// TwinCAT 3 PLC project Pinana
// Title: Pinanas
// Company: ekvip automation GmbH
// Author: Ajnin and Yeknom
// Description: short summary ============= This project was created for the YouTube channel https://www.youtube.com/@ninjamonkeystutorials created. It is intended to show why references as return values for functions are dangerous. legal notes ======== SPDX-FileCopyrightText: © 2024 ekvip automation GmbH <info@ekvip.de> SPDX-License-Identifier: Apache-2.0 For details check: Apache-2.0_
// ProgramVersion: 3.1.4024.0
// libraries:
//   Tc2_Standard, * (Beckhoff Automation GmbH)
//   Tc2_System, * (Beckhoff Automation GmbH)
//   Tc3_Module, * (Beckhoff Automation GmbH)
// project tree:
//   Pinana/Banana/Types/Enums/ BananaType.TcDUT
//   Pinana/Functions/ CalculatePinanaCurvature.TcPOU, GetANewPinana.TcPOU, GetAPinana.TcPOU, GetAPinanaFromGlobal.TcPOU, GetAPinanaFromStack.TcPOU, IsSetPinanaCallByRef.TcPOU
//   Pinana/GVLs/ PinanaPrototypes.TcGVL
//   Pinana/Pineapple/Types/Enums/ PineappleType.TcDUT
//   Pinana/Types/Enums/ PinanaType.TcDUT
//   Pinana/Types/Structures/ Pinana.TcDUT
//   Tasks/main/ MAIN.TcPOU, PlcTask.TcTTO
// real-time tasks:
//   TASK PlcTask: cycle T#10ms, priority 20, ADS port 350

CONFIGURATION Pinana
    RESOURCE PLC ON TwinCAT3
        TASK PlcTask(INTERVAL := T#10ms, PRIORITY := 20);
        PROGRAM MAIN WITH PlcTask : MAIN;
    END_RESOURCE
END_CONFIGURATION

// ---- Pinana/Banana/Types/Enums/BananaType.TcDUT
(*

short summary
=============
This enumeration represents the banana varieties from which π-nana are to be produced.
If the type is extended, make sure that only the least significant nibble is used.
Only 15 banana types can be mapped, namely from 16#01 to 16#0F.
The software generates the π-nana type by adding the pineapple type and the banana type.
So that everything remains unique, the pineapple variety is given the second nibble from 16#10 to 16#F0.

legal notes
===========
SPDX-FileCopyrightText: © 2024 ekvip automation GmbH <info@ekvip.de>
SPDX-License-Identifier: Apache-2.0
For details check: Apache-2.0_

.. _Apache-2.0: https://www.apache.org/licenses/LICENSE-2.0

*)
{attribute 'qualified_only'}
{attribute 'strict'}
{attribute 'to_string'}
TYPE BananaType :(
	(* it's not a banana *)
	NONE		:= 16#00,
	(* it's a cavendish banana *)
	CAVENDISH	:= 16#01,
	(* it's a plaintain banana *)
	PLANTAIN	:= 16#02,
	(* it's a red banana *)
	RED_BANANA	:= 16#03,
	(* it's a lady finger banana and not an okra *)
	LADY_FINGER	:= 16#04
)UDINT := NONE;
END_TYPE

// ---- Pinana/Pineapple/Types/Enums/PineappleType.TcDUT
(*

short summary
=============
This enumeration represents the pineapple varieties from which π-nana are to be produced.
If the type is extended, make sure that only the second nibble is used.
Only 15 pineapple types can be mapped, namely from 16#10 to 16#F0.
The software generates the π-nana type by adding the pineapple type and the banana type.
So that everything remains unique, the banana variety is given the least significant nibble from 16#01 to 16#0F.


legal notes
===========
SPDX-FileCopyrightText: © 2024 ekvip automation GmbH <info@ekvip.de>
SPDX-License-Identifier: Apache-2.0
For details check: Apache-2.0_

.. _Apache-2.0: https://www.apache.org/licenses/LICENSE-2.0

*)
{attribute 'qualified_only'}
{attribute 'strict'}
{attribute 'to_string'}
TYPE PineappleType :(
	(* it's not a pineapple *)
	NONE		:= 16#00,
	(* it's an abacaxi pineapple *)
	ABACAXI		:= 16#10,
	(* it's a queen pineapple *)
	QUEEN		:= 16#20,
	(* it's a mordilona pineapple *)
	MORDILONA	:= 16#30,
	(* it's a panare pineapple *)
	PANARE		:= 16#40
)UDINT := NONE;
END_TYPE

// ---- Pinana/Types/Enums/PinanaType.TcDUT
(*

short summary
=============
This enumeration represents the π-nana types.
The type of π-nana is determined by the simple formula
π-nana type := pineapple type + banana type 

legal notes
===========
SPDX-FileCopyrightText: © 2024 ekvip automation GmbH <info@ekvip.de>
SPDX-License-Identifier: Apache-2.0
For details check: Apache-2.0_

.. _Apache-2.0: https://www.apache.org/licenses/LICENSE-2.0

*)
{attribute 'qualified_only'}
{attribute 'to_string'}
TYPE PinanaType :
(
	(* it's not a pinana *)
	NONE		:= 16#00,
	(* PineappleType.ABACAXI + BananaType.CAVENDISH *)
	ABADISH 	:= 16#11,
	(* PineappleType.ABACAXI + BananaType.PLANTAIN *)
	PLANABA		:= 16#12,
	(* PineappleType.ABACAXI + BananaType.RED_BANANA *)
	ABANANA		:= 16#13,
	(* PineappleType.ABACAXI + BananaType.LADY_FINGER *)
	ABA_LADY	:= 16#14,
	(* PineappleType.QUEEN + BananaType.CAVENDISH *)
	CAVEEN	 	:= 16#21,
	(* PineappleType.QUEEN + BananaType.PLANTAIN *)
	PLEEN		:= 16#22,
	(* PineappleType.QUEEN + BananaType.RED_BANANA *)
	RED_QUEEN	:= 16#23,
	(* PineappleType.QUEEN + BananaType.LADY_FINGER *)
	LADY_QUEEN	:= 16#24,
	(* PineappleType.MORDILONA + BananaType.CAVENDISH *)
	ILONACAVE 	:= 16#31,
	(* PineappleType.MORDILONA + BananaType.PLANTAIN *)
	PLAONA		:= 16#32,
	(* PineappleType.MORDILONA + BananaType.RED_BANANA *)
	RED_LONA	:= 16#33,
	(* PineappleType.MORDILONA + BananaType.LADY_FINGER *)
	LADY_LONA	:= 16#34,
	(* PineappleType.PANARE + BananaType.CAVENDISH *)
	PANDISH 	:= 16#41,
	(* PineappleType.PANARE + BananaType.PLANTAIN *)
	PLANPAN		:= 16#42,
	(* PineappleType.PANARE + BananaType.RED_BANANA *)
	PANANA		:= 16#43,
	(* PineappleType.PANARE + BananaType.LADY_FINGER *)
	PAN_FINGER	:= 16#44	
)UDINT := NONE;
END_TYPE

// ---- Pinana/Types/Structures/Pinana.TcDUT
(*

short summary
=============
This type struct contains the properties of a π-nana.

legal notes
===========
SPDX-FileCopyrightText: © 2024 ekvip automation GmbH <info@ekvip.de>
SPDX-License-Identifier: Apache-2.0
For details check: Apache-2.0_

.. _Apache-2.0: https://www.apache.org/licenses/LICENSE-2.0

*)
TYPE Pinana :
STRUCT
	(* pointer to itself for destruction of dynamically created Pinanas *)
	me			:POINTER TO Pinana := 0;
	(* type of π-nana *)
	pinanaType	:PinanaType;
	(* name of the π-nana variety *)
	variety		:STRING;
	(* curvature of π-nana ofcourse in radians *)
	curve		:LREAL;
END_STRUCT
END_TYPE

// ---- Pinana/GVLs/PinanaPrototypes.TcGVL
(*

short summary
=============
This is a lookup table for π-nanas.
It's not a constant because the function GetAPinanaFromGlobal
has a reference to π-nana as return value. A reference requires write access.

The attribute hide is not used because we want show it online how to screw it. 

legal notes
===========
SPDX-FileCopyrightText: © 2024 ekvip automation GmbH <info@ekvip.de>
SPDX-License-Identifier: Apache-2.0
For details check: Apache-2.0_

.. _Apache-2.0: https://www.apache.org/licenses/LICENSE-2.0

*)
{attribute 'qualified_only'}
VAR_GLOBAL
	(* lookup table for π-nanas *)
	pinanas :ARRAY[
		SHR(PineappleType.ABACAXI,4)..SHR(PineappleType.PANARE,4)
	] OF ARRAY[
		BananaType.CAVENDISH..BananaType.LADY_FINGER
	] OF Pinana := [
		[
			(pinanaType := PinanaType.ABADISH,		variety := TO_STRING(PinanaType.ABADISH),	curve := CalculatePinanaCurvature(PinanaType.ABADISH),		me := ADR(pinanas[1][1])),
			(pinanaType := PinanaType.PLANABA,		variety := TO_STRING(PinanaType.PLANABA),	curve := CalculatePinanaCurvature(PinanaType.PLANABA),		me := ADR(pinanas[1][2])),
			(pinanaType := PinanaType.ABANANA,		variety := TO_STRING(PinanaType.ABANANA),	curve := CalculatePinanaCurvature(PinanaType.ABANANA),		me := ADR(pinanas[1][3])),
			(pinanaType := PinanaType.ABA_LADY,		variety := TO_STRING(PinanaType.ABA_LADY),	curve := CalculatePinanaCurvature(PinanaType.ABA_LADY),		me := ADR(pinanas[1][4]))
		],[
			(pinanaType := PinanaType.CAVEEN,		variety := TO_STRING(PinanaType.CAVEEN),	curve := CalculatePinanaCurvature(PinanaType.CAVEEN),		me := ADR(pinanas[2][1])),
			(pinanaType := PinanaType.PLEEN,		variety := TO_STRING(PinanaType.PLEEN),		curve := CalculatePinanaCurvature(PinanaType.PLEEN),		me := ADR(pinanas[2][2])),
			(pinanaType := PinanaType.RED_QUEEN,	variety := TO_STRING(PinanaType.RED_QUEEN),	curve := CalculatePinanaCurvature(PinanaType.RED_QUEEN),	me := ADR(pinanas[2][3])),
			(pinanaType := PinanaType.LADY_QUEEN,	variety := TO_STRING(PinanaType.LADY_QUEEN),curve := CalculatePinanaCurvature(PinanaType.LADY_QUEEN),	me := ADR(pinanas[2][4]))
		],[
			(pinanaType := PinanaType.ILONACAVE,	variety := TO_STRING(PinanaType.ILONACAVE),	curve := CalculatePinanaCurvature(PinanaType.ILONACAVE),	me := ADR(pinanas[3][1])),
			(pinanaType := PinanaType.PLAONA,		variety := TO_STRING(PinanaType.PLAONA),	curve := CalculatePinanaCurvature(PinanaType.PLAONA),		me := ADR(pinanas[3][2])),
			(pinanaType := PinanaType.RED_LONA,		variety := TO_STRING(PinanaType.RED_LONA),	curve := CalculatePinanaCurvature(PinanaType.RED_LONA),		me := ADR(pinanas[3][3])),
			(pinanaType := PinanaType.LADY_LONA,	variety := TO_STRING(PinanaType.LADY_LONA),	curve := CalculatePinanaCurvature(PinanaType.LADY_LONA),	me := ADR(pinanas[3][4]))
		],[
			(pinanaType := PinanaType.PANDISH,		variety := TO_STRING(PinanaType.PANDISH),	curve := CalculatePinanaCurvature(PinanaType.PANDISH),		me := ADR(pinanas[4][1])),
			(pinanaType := PinanaType.PLANPAN,		variety := TO_STRING(PinanaType.PLANPAN),	curve := CalculatePinanaCurvature(PinanaType.PLANPAN),		me := ADR(pinanas[4][2])),
			(pinanaType := PinanaType.PANANA,		variety := TO_STRING(PinanaType.PANANA),	curve := CalculatePinanaCurvature(PinanaType.PANANA),		me := ADR(pinanas[4][3])),
			(pinanaType := PinanaType.PAN_FINGER,	variety := TO_STRING(PinanaType.PAN_FINGER),curve := CalculatePinanaCurvature(PinanaType.PAN_FINGER),	me := ADR(pinanas[4][4]))
		]
	];
END_VAR

// ---- Tasks/main/MAIN.TcPOU
(*

short summary
=============
This program is attached to the main plc task.
This project was created for the YouTube channel https://www.youtube.com/@ninjamonkeystutorials
created. It is intended to show why references as return values for functions are dangerous.
You've a couple of flags to control the data flow... 
It can be a lot of fun to mess with TwinCAT, if it's not a real world plc. So have fun with it.

legal notes
===========
SPDX-FileCopyrightText: © 2024 ekvip automation GmbH <info@ekvip.de>
SPDX-License-Identifier: Apache-2.0
For details check: Apache-2.0_

.. _Apache-2.0: https://www.apache.org/licenses/LICENSE-2.0

*)
PROGRAM MAIN
VAR
	//set it in online mode to skip all methods
	skipAll				:BOOL := FALSE;
	//set it in online mode to skip no method, but skipAll must be unset
	skipNone			:BOOL := FALSE;
	//unset it in online mode if you want to step through messWithGlobalPinanas, but skipAll must be unset
	skipMessWithGlobal	:BOOL := TRUE;
	//unset it in online mode if you want to step through messWithNewPinanas, but skipAll must be unset
	skipMessWithNew		:BOOL := TRUE;
	//unset it in online mode if you want to step through messWithStackPinanas, but skipAll must be unset
	skipMessWithStack	:BOOL := TRUE;
	//unset it in online mode if you want to step through withCallByRef, but skipAll must be unset
	skipCallByRef		:BOOL := TRUE;
	//unset it in online mode if you want to step through withACommonReturn, but skipAll must be unset
	skipCommon			:BOOL := TRUE;
	//reference to our π-nana from stack
	stackPinana			:REFERENCE TO Pinana;
	//reference to our π-nana from the global variable list
	globalPinana		:REFERENCE TO Pinana;
	//reference to our new π-nana
	newPinana			:REFERENCE TO Pinana;
END_VAR

messWithStackPinanas(isSkipIt(skipMessWithStack));
messWithGlobalPinanas(isSkipIt(skipMessWithGlobal));
messWithNewPinanas(isSkipIt(skipMessWithNew));
withCallByRef(isSkipIt(skipCallByRef));
withACommonReturn(isSkipIt(skipCommon));

(*

short summary
=============
This method returns TRUE if a skip is required.

legal notes
===========
SPDX-FileCopyrightText: © 2024 ekvip automation GmbH <info@ekvip.de>
SPDX-License-Identifier: Apache-2.0
For details check: Apache-2.0_

.. _Apache-2.0: https://www.apache.org/licenses/LICENSE-2.0

*)
METHOD isSkipIt :BOOL
VAR_INPUT
	(* specific skipping flag to check *)
	skip	:BOOL;
END_VAR
isSkipIt := skipAll;
RETURN(skipAll);
isSkipIt := (NOT skipNone);
RETURN(skipNone);
isSkipIt := skip;
END_METHOD

(*

short summary
=============
This method exploids the reference return value of the function GetAPinanaFromGlobal
Use break points to check it out by your self.

legal notes
===========
SPDX-FileCopyrightText: © 2024 ekvip automation GmbH <info@ekvip.de>
SPDX-License-Identifier: Apache-2.0
For details check: Apache-2.0_

.. _Apache-2.0: https://www.apache.org/licenses/LICENSE-2.0

*)
METHOD messWithGlobalPinanas
VAR_INPUT
	(* flag to skip this method *)
	skip	:BOOL;
END_VAR
VAR
	(* a π-nana type to fetch it from GetAPinanaFromGlobal *)
	typeOfPinana	:PinanaType;
	(* a π-nana to fetch it from GetAPinanaFromGlobal *)
	pinana			:Pinana;
	(* π-nana varity to fetch it from GetAPinanaFromGlobal *)
	name			:STRING;
	(* set it true to get exception from using an invalid reference *)
	skipException	:BOOL := TRUE;
END_VAR
RETURN(skip);
//every thing is fine here
pinana := GetAPinanaFromGlobal(PineappleType.QUEEN, BananaType.RED_BANANA);
name := pinana.variety; //RED_QUEEN
name := GetAPinanaFromGlobal(PineappleType.QUEEN, BananaType.LADY_FINGER).variety; //LADY_QUEEN


globalPinana REF= GetAPinanaFromGlobal(PineappleType.QUEEN, BananaType.RED_BANANA);
RETURN(NOT __ISVALIDREF(globalPinana));
name := globalPinana.variety; //RED_QUEEN
name := GetAPinanaFromGlobal(PineappleType.QUEEN, BananaType.RED_BANANA).variety; //RED_QUEEN

globalPinana.variety := 'Gold Kiwi'; // here we overwrite the global variable, and this is hard to find
name := GetAPinanaFromGlobal(PineappleType.QUEEN, BananaType.RED_BANANA).variety; //RED_QUEEN is expected but we get Gold Kiwi
globalPinana.variety := TO_STRING(pinana.pinanaType);// here we overwrite the global variable again to the old value

//unset skipException if you want a exception
JMP(skipException) END;
typeOfPinana := GetAPinanaFromGlobal(PineappleType.NONE, BananaType.NONE).pinanaType;

END:
END_METHOD

(*

short summary
=============
This method exploids the reference return value of the function GetANewPinana
Use break points to check it out by your self.

legal notes
===========
SPDX-FileCopyrightText: © 2024 ekvip automation GmbH <info@ekvip.de>
SPDX-License-Identifier: Apache-2.0
For details check: Apache-2.0_

.. _Apache-2.0: https://www.apache.org/licenses/LICENSE-2.0

*)
METHOD messWithNewPinanas
VAR_INPUT
	(* flag to skip this method *)
	skip	:BOOL;
END_VAR
VAR
	(* a π-nana type to fetch it from GetANewPinana *)
	typeOfPinana	:PinanaType;
	(* a π-nana to fetch it from GetANewPinana *)
	pinana			:Pinana;
	(* π-nana varity to fetch it from GetANewPinana *)
	name			:STRING;
	(* set it true to get exception from using an invalid reference *)
	skipException	:BOOL := TRUE;
	(* byte pointer to free the new π-nana again *)
	void			:POINTER TO BYTE;
END_VAR
RETURN(skip);
//here is everthing fine
newPinana REF= GetANewPinana(PineappleType.QUEEN, BananaType.RED_BANANA);
RETURN(NOT __ISVALIDREF(newPinana));
name := newPinana.variety; //RED_QUEEN
//clean up again
void := newPinana.me;
__DELETE(void);
//normaly we should delete the reference again
//newPinana REF= 0;

pinana := GetANewPinana(PineappleType.QUEEN, BananaType.LADY_FINGER);
name := pinana.variety; //LADY_QUEEN
//clean up again
void := pinana.me;
__DELETE(void);
pinana.me := 0;
pinana.curve := 0;
pinana.pinanaType := PinanaType.NONE;
pinana.variety := TO_STRING(PinanaType.NONE);

//how to get a memory leak because we are not able to clean up the memory anymore
name := GetANewPinana(PineappleType.QUEEN, BananaType.RED_BANANA).variety; //RED_QUEEN

//unset skipException if you want a exception
JMP(skipException) END;
typeOfPinana := GetAPinanaFromGlobal(PineappleType.NONE, BananaType.NONE).pinanaType;

END:
END_METHOD

(*

short summary
=============
This method exploids the reference return value of the function GetAPinanaFromStack
Use break points to check it out by your self.

legal notes
===========
SPDX-FileCopyrightText: © 2024 ekvip automation GmbH <info@ekvip.de>
SPDX-License-Identifier: Apache-2.0
For details check: Apache-2.0_

.. _Apache-2.0: https://www.apache.org/licenses/LICENSE-2.0

*)
METHOD messWithStackPinanas
VAR_INPUT
	(* flag to skip this method *)
	skip	:BOOL;
END_VAR
VAR
	(* a π-nana type to fetch it from GetAPinanaFromStack *)
	typeOfPinana	:PinanaType;
	(* a π-nana to fetch it from GetAPinanaFromStack *)
	pinana			:Pinana;
	(* π-nana varity to fetch it from GetAPinanaFromStack *)
	name			:STRING;
	(* set it true to get exception from using an invalid reference *)
	skipException	:BOOL := TRUE;
END_VAR
RETURN(skip);
//every thing is fine here
pinana := GetAPinanaFromStack(PineappleType.QUEEN, BananaType.RED_BANANA);
name := pinana.variety; //RED_QUEEN
name := GetAPinanaFromStack(PineappleType.QUEEN, BananaType.LADY_FINGER).variety; //LADY_QUEEN

//we create now a valid reference but it points to the stack
stackPinana REF= GetAPinanaFromStack(PineappleType.QUEEN, BananaType.RED_BANANA);
RETURN(NOT __ISVALIDREF(stackPinana));
name := stackPinana.variety; //RED_QUEEN is expected
name := GetAPinanaFromStack(PineappleType.QUEEN, BananaType.RED_BANANA).variety; //RED_QUEEN

//dangerous: here we try to overwrite the stack memory. To see the problem run it more than once
//stackPinana.variety := 'Gold Kiwi';
//dangerous: here we overwrite the stack memory
//stackPinana.me^.variety := 'banana phone';

//unset skipException if you want a exception
JMP(skipException) END;
typeOfPinana := GetAPinanaFromStack(PineappleType.NONE, BananaType.NONE).pinanaType;

END:
END_METHOD

(*

short summary
=============
This method is just to show, there is nothing to exploid with a common return

legal notes
===========
SPDX-FileCopyrightText: © 2024 ekvip automation GmbH <info@ekvip.de>
SPDX-License-Identifier: Apache-2.0
For details check: Apache-2.0_

.. _Apache-2.0: https://www.apache.org/licenses/LICENSE-2.0

*)
METHOD withACommonReturn
VAR_INPUT
	(* flag to skip this method *)
	skip	:BOOL;
END_VAR
VAR
	(* a π-nana to fetch it from GetAPinana *)
	pinana			:Pinana;
	(* π-nana varity to fetch it from GetAPinana *)
	name			:STRING;
END_VAR
RETURN(skip);
//every thing is fine here
pinana := GetAPinana(PineappleType.QUEEN, BananaType.RED_BANANA);
name := pinana.variety; //RED_QUEEN
pinana := GetAPinana(PineappleType.NONE, BananaType.NONE);
name := pinana.variety; //NONE
END_METHOD

(*

short summary
=============
his method is just to show, it's safer with a call by reference

legal notes
===========
SPDX-FileCopyrightText: © 2024 ekvip automation GmbH <info@ekvip.de>
SPDX-License-Identifier: Apache-2.0
For details check: Apache-2.0_

.. _Apache-2.0: https://www.apache.org/licenses/LICENSE-2.0

*)
METHOD withCallByRef
VAR_INPUT
	(* flag to skip this method *)
	skip	:BOOL;
END_VAR
VAR
	(* a π-nana to fetch it from IsSetPinanaCallByRef *)
	pinana			:Pinana;
	(* π-nana varity to fetch it from IsSetPinanaCallByRef *)
	name			:STRING;
	(* π-nana address to show the equality *)
	{attribute 'displaymode':='hex'}
	pinanaAddress	:__UXINT;
	(* π-nana address to show the equality *)
	{attribute 'displaymode':='hex'}
	meAddress		:__UXINT;
END_VAR
RETURN(skip);
//every thing is fine
IsSetPinanaCallByRef(PineappleType.QUEEN, BananaType.RED_BANANA, pinana);
name := pinana.variety; //RED_QUEEN

//check the addresses
pinanaAddress := ADR(pinana);
meAddress := pinana.me;
IF (pinanaAddress = meAddress) THEN
	name := 'Addresses are equal';
END_IF

(*
it's impossible to run code like below 
because it's not compileable 
so you can't throw an exception

IsSetPinanaCallByRef(
	pineapple := PineappleType.QUEEN,
	banana := BananaType.RED_BANANA,
	pinana := 0
);
*)

IF (NOT IsSetPinanaCallByRef(PineappleType.NONE, BananaType.NONE, pinana)) THEN
	name := pinana.variety;
	;//Error handling here
END_IF
END_METHOD

END_PROGRAM

// ---- Pinana/Functions/GetAPinanaFromGlobal.TcPOU
(*

short summary
=============
This function returns a reference to a π-nana.
The reference is created by a pineapple type and a banana type.
The reference points to a π-nana of the global lookup table PinanaPrototypes.pinanas.

legal notes
===========
SPDX-FileCopyrightText: © 2024 ekvip automation GmbH <info@ekvip.de>
SPDX-License-Identifier: Apache-2.0
For details check: Apache-2.0_

.. _Apache-2.0: https://www.apache.org/licenses/LICENSE-2.0

*)
FUNCTION GetAPinanaFromGlobal :REFERENCE TO Pinana
VAR_INPUT
	(* type of pineapple to create a π-nana from it *)
	pineapple	:PineappleType;
	(* type of banana to create a π-nana from it *)
	banana		:BananaType;
END_VAR

GetAPinanaFromGlobal REF= 0;
RETURN((pineapple = PineappleType.NONE) OR (banana = BananaType.NONE));
GetAPinanaFromGlobal REF= PinanaPrototypes.pinanas[SHR(pineapple,4)][banana];

END_FUNCTION

// ---- Pinana/Functions/GetANewPinana.TcPOU
(*

short summary
=============
This function dynamically allocates memory and thus creates a new π-nana from a pineapple type and a banana type.
The pointer pinana.me specifies the address of the new π-nana to free it again later.
The π-nana allocates the memory as a byte, as π-nanas do not have the enable dynamic creation attribute.
It returns a reference to the new π-nana.

legal notes
===========
SPDX-FileCopyrightText: © 2024 ekvip automation GmbH <info@ekvip.de>
SPDX-License-Identifier: Apache-2.0
For details check: Apache-2.0_

.. _Apache-2.0: https://www.apache.org/licenses/LICENSE-2.0

*)
FUNCTION GetANewPinana :REFERENCE TO Pinana
VAR_INPUT
	(* type of pineapple to create a π-nana from it *)
	pineapple	:PineappleType;
	(* type of banana to create a π-nana from it *)
	banana		:BananaType;
END_VAR
VAR
	(* byte pointer to allocate the memory for the new π-nana *)
	bytePointer		:POINTER TO BYTE;
	(* pointer to the new created π-nana *) 
	pinanaPointer	:POINTER TO Pinana;
END_VAR
VAR CONSTANT
	(* just a null pointer address *)
	{attribute 'const_replaced'}
	NULL 		:__XWORD := 0;
END_VAR

GetANewPinana REF= 0;
(* validate parameters *)
RETURN((pineapple = PineappleType.NONE) OR (banana = BananaType.NONE));
(* allocate memory for the new π-nana *)
bytePointer := __NEW(BYTE, SIZEOF(Pinana));
RETURN(bytePointer = NULL);
(* initialize new π-nana *)
pinanaPointer := bytePointer;
pinanaPointer^.me := bytePointer;
pinanaPointer^.pinanaType := (TO_UDINT(pineapple) + TO_UDINT(banana));
pinanaPointer^.variety := TO_STRING(pinanaPointer^.pinanaType);
pinanaPointer^.curve := CalculatePinanaCurvature(pinanaPointer^.pinanaType);
GetANewPinana REF= pinanaPointer^;

END_FUNCTION

// ---- Pinana/Functions/CalculatePinanaCurvature.TcPOU
(*

short summary
=============
This function returns the curvature of a π-nana.
It uses the function block Tc2_System.DRAND and the π-nana type is used as the seed.
As the function block is on the stack, Tc2_System.DRAND should return the same value for each π-nana type.
A lookup table would have been a better choice, but less fancy.
The curvature of the π-nana is not specified in degrees but in radians.

legal notes
=================
SPDX-FileCopyrightText: © 2024 ekvip automation GmbH <info@ekvip.de>
SPDX-License-Identifier: Apache-2.0
For details check: Apache-2.0_

.. _Apache-2.0: https://www.apache.org/licenses/LICENSE-2.0

*)
FUNCTION CalculatePinanaCurvature :LREAL
VAR_INPUT
	(* type of the π-nana to calculate the curvature for it *)
	typeOfPinana :PinanaType;
END_VAR
VAR
	(* random number generator, it generates no random numbers because it's on the stack *)
	rand		:Tc2_System.DRAND;
END_VAR
VAR CONSTANT
	(* an approximation of the circle number pi *)
	PI	 		:REAL := 3.14159265359;
	(* just 180 degree *)
	SEMICIRCLE	:REAL := 180.0;
END_VAR

CalculatePinanaCurvature := 0.0;
RETURN(typeOfPinana = PinanaType.NONE);
rand(Seed := TO_INT(typeOfPinana));
CalculatePinanaCurvature := (
	(
		TO_REAL(
			TO_ULINT(
				TO_REAL(rand.Num) * 1.0E+6
			) MOD 30
		) + TO_REAL(rand.Num)
	) * (PI/SEMICIRCLE)
);

END_FUNCTION

// ---- Pinana/Functions/GetAPinanaFromStack.TcPOU
(*

short summary
=============
This function returns a reference to a π-nana.
The π-nana is created by a pineapple type and a banana type.
The reference points to a π-nana on the stack memory.

legal notes
===========
SPDX-FileCopyrightText: © 2024 ekvip automation GmbH <info@ekvip.de>
SPDX-License-Identifier: Apache-2.0
For details check: Apache-2.0_

.. _Apache-2.0: https://www.apache.org/licenses/LICENSE-2.0

*)
FUNCTION GetAPinanaFromStack :REFERENCE TO Pinana
VAR_INPUT
	(* type of pineapple to create a π-nana from it *)
	pineapple	:PineappleType;
	(* type of banana to create a π-nana from it *)
	banana		:BananaType;
END_VAR
VAR
	(* stack π-nana to refer on it *)
	stackPinana :Pinana;
END_VAR

GetAPinanaFromStack REF= 0;
(* validate parameters *)
RETURN((pineapple = PineappleType.NONE) OR (banana = BananaType.NONE));

(* initialize stack π-nana *)
stackPinana.me := ADR(stackPinana);
stackPinana.pinanaType := (TO_UDINT(pineapple) + TO_UDINT(banana));
stackPinana.variety := TO_STRING(stackPinana.pinanaType);
stackPinana.curve := CalculatePinanaCurvature(stackPinana.pinanaType);
GetAPinanaFromStack REF= stackPinana;

END_FUNCTION

// ---- Pinana/Functions/GetAPinana.TcPOU
(*

short summary
=============
This function returns a π-nana from a pineapple type and a banana type.

legal notes
===========
SPDX-FileCopyrightText: © 2024 ekvip automation GmbH <info@ekvip.de>
SPDX-License-Identifier: Apache-2.0
For details check: Apache-2.0_

.. _Apache-2.0: https://www.apache.org/licenses/LICENSE-2.0

*)
FUNCTION GetAPinana :Pinana
VAR_INPUT
	(* type of pineapple to create a π-nana from it *)
	pineapple	:PineappleType;
	(* type of banana to create a π-nana from it *)
	banana		:BananaType;
END_VAR
VAR CONSTANT
	(* just a null pointer address *)
	{attribute 'const_replaced'}
	NULL 		:__XWORD := 0;
END_VAR

(* validate parameters *)
RETURN((pineapple = PineappleType.NONE) OR (banana = BananaType.NONE));

(* initialize π-nana *)
GetAPinana.me := NULL;
GetAPinana.pinanaType := (TO_UDINT(pineapple) + TO_UDINT(banana));
GetAPinana.variety := TO_STRING(GetAPinana.pinanaType);
GetAPinana.curve := CalculatePinanaCurvature(GetAPinana.pinanaType);

END_FUNCTION

// ---- Pinana/Functions/IsSetPinanaCallByRef.TcPOU
(*

short summary
=============
This function sets the content of a π-nana by a pineapple type and a banana type.
It returns true if it was successful and 
false if it can't deterime a π-nana of type pineapple and banana.
The function clears the old π-nana content in every case.

legal notes
===========
SPDX-FileCopyrightText: © 2024 ekvip automation GmbH <info@ekvip.de>
SPDX-License-Identifier: Apache-2.0
For details check: Apache-2.0_

.. _Apache-2.0: https://www.apache.org/licenses/LICENSE-2.0

*)
FUNCTION IsSetPinanaCallByRef :BOOL
VAR_INPUT
	(* type of pineapple to get a π-nana from it *)
	pineapple	:PineappleType;
	(* type of banana to get a π-nana from it *)
	banana		:BananaType;
END_VAR
VAR_IN_OUT
	(* reference to a π-nana to set it*)
	pinanaToSet 	:Pinana;	
END_VAR
VAR CONSTANT
	(* null byte to clear the old π-nana content *) 
	{attribute 'const_replaced'}
	NULL 		:USINT := 0;
END_VAR

IsSetPinanaCallByRef := FALSE;
Tc2_System.MEMSET(ADR(pinanaToSet), NULL, SIZEOF(Pinana));
pinanaToSet.variety := TO_STRING(PinanaType.NONE);
(* validate parameters *)
RETURN((pineapple = PineappleType.NONE) OR (banana = BananaType.NONE));

(* set new π-nana content *)
pinanaToSet.me := ADR(pinanaToSet);
pinanaToSet.pinanaType := (TO_UDINT(pineapple) + TO_UDINT(banana));
pinanaToSet.variety := TO_STRING(pinanaToSet.pinanaType);
pinanaToSet.curve := CalculatePinanaCurvature(pinanaToSet.pinanaType);
IsSetPinanaCallByRef := TRUE;

END_FUNCTION
